// TwinCAT 3 PLC project SH_FileReader
// Title: SH_FileReader
// Company: Stefan Halder
// ProjectVersion: 1.0.0.0
// ProgramVersion: 3.1.4026.12
// libraries:
//   Tc2_Standard, * (Beckhoff Automation GmbH)
//   Tc2_System, * (Beckhoff Automation GmbH)
//   Tc2_Utilities, * (Beckhoff Automation GmbH)
// project tree:
//   FileReader/DUTs/ ERROR.TcDUT, STATE.TcDUT (not stored)
//   FileReader/ FileReader.TcPOU
// real-time tasks:
//   TASK PlcTask: cycle T#10ms, priority 20, ADS port 350

// ---- FileReader/DUTs/ERROR.TcDUT
TYPE ERROR :
STRUCT
	bError : BOOL;
	nErrorCode : DINT;
END_STRUCT
END_TYPE

// ---- FileReader/FileReader.TcPOU
FUNCTION_BLOCK FileReader
VAR CONSTANT
	iC_MAX_NUM_LINES_IN_FILE : UINT := 1000;
	iC_MAX_STRING_LENGTH : UINT := 25;
END_VAR
VAR
	_bBusy : BOOL;
	_sFilePath : STRING;
	_arsFileContent : ARRAY [0..iC_MAX_NUM_LINES_IN_FILE] OF STRING(iC_MAX_STRING_LENGTH);
	
	fbi_FileOpen : FB_FileOpen;
	fbi_FileGets : FB_FileGets;
	fbi_FileClose : FB_FileClose;
	
	eState : STATE := STATE.Idle;
	
	hFileHandle : UINT;
	iFileContentNextIndex : UINT;
	stError : ERROR;
END_VAR

CASE eState OF
	State.Idle:
		// Do nothing
	State.OpenFile:
		_bBusy := TRUE;
		iFileContentNextIndex := 0;
		MEMSET(ADR(_arsFileContent), 0, SIZEOF(_arsFileContent));
		fbi_FileOpen(sPathName := sFilePath, nMode := FOPEN_MODEREAD OR FOPEN_MODETEXT, ePath := PATH_GENERIC, bExecute := TRUE, bError => stError.bError, nErrId => stError.nErrorCode);
		eState := STATE.OpenFileAwaitFinish;
		
	State.OpenFileAwaitFinish:
		fbi_FileOpen(bExecute := FALSE, hFile => hFileHandle, bError => stError.bError, nErrId => stError.nErrorCode);
		IF NOT fbi_FileOpen.bBusy THEN
			IF NOT stError.bError THEN
				eState := STATE.ReadFile;
			ELSE
				eState := STATE.Error;
			END_IF
		END_IF
		
	State.ReadFile:
		fbi_FileGets(hFile := hFileHandle, bExecute := TRUE, bError => stError.bError, nErrId => stError.nErrorCode);
		eState := STATE.ReadFileAwaitFinish;
		
	State.ReadFileAwaitFinish:
		fbi_FileGets(bExecute := FALSE, bError => stError.bError, nErrId => stError.nErrorCode);
		IF NOT fbi_FileGets.bBusy THEN
			IF NOT stError.bError THEN
				_arsFileContent[iFileContentNextIndex] := fbi_FileGets.sLine;
				IF fbi_FileGets.bEOF THEN
					eState := STATE.CloseFile;
				ELSE
					eState := STATE.ReadFile;
					iFileContentNextIndex := iFileContentNextIndex+1;	
				END_IF
			ELSE
				eState := STATE.Error;
			END_IF	
		END_IF
		
	State.CloseFile:
		fbi_FileClose(hFile := hFileHandle, bExecute := TRUE, bError => stError.bError, nErrId => stError.nErrorCode);
		eState := STATE.CloseFileAwaitFinish;
		
	State.CloseFileAwaitFinish:
		fbi_FileClose(bExecute := FALSE, bError => stError.bError, nErrId => stError.nErrorCode);
		IF NOT fbi_FileClose.bBusy THEN
			IF NOT stError.bError THEN
				eState := STATE.Idle;
			ELSE
				eState := STATE.Error;
			END_IF
			_bBusy := FALSE;
			hFileHandle := 0;
		END_IF
		
	State.Error:
		eState := STATE.Idle;
END_CASE

PROPERTY arsFileContent : ARRAY [0..iC_MAX_NUM_LINES_IN_FILE] OF STRING(iC_MAX_STRING_LENGTH)
GET
arsFileContent := _arsFileContent;
END_GET
END_PROPERTY

PROPERTY bBusy : BOOL
GET
bBusy := _bBusy;
END_GET
END_PROPERTY

METHOD GetLineByIndex : STRING
VAR_INPUT
	iIndex : UINT;
END_VAR
GetLineByIndex := _arsFileContent[iIndex];
END_METHOD

METHOD ReadFile : BOOL
VAR_INPUT
	bExecute : BOOL;
	sFilePath : STRING;
END_VAR
VAR_OUTPUT
	stError : ERROR;
END_VAR
VAR
	bExecute_RTrig : R_TRIG;
END_VAR
_sFilePath := sFilePath;
bExecute_RTrig(CLK := bExecute);
IF bExecute_RTRIG.Q THEN
	IF eState = STATE.Idle THEN
		_bBusy := TRUE;
		eState := STATE.OpenFile;
		stError.bError := FALSE;
		stError.nErrorCode := 0;
	ELSE
		stError.bError := TRUE;
		stError.nErrorCode := 1; //FB not ready		
	END_IF
END_IF
ReadFile := NOT _bBusy OR stError.bError;
END_METHOD

PROPERTY sFilePath : STRING
GET
sFilePath := _sFilePath;
END_GET
SET
_sFilePath := sFilePath;
END_SET
END_PROPERTY

END_FUNCTION_BLOCK
